PROGRAM MAIN
VAR
	test : UINT;
END_VAR


//DAQ test
//fssf

//daq test

//One

//Two

//Threee


//Four 

//Five

//Six


//Seven

//Eight


//Nine

//Ten

END_PROGRAM

(* stored: Version 1.1.0.1, ProductVersion 3.1.4024.9
   POU MAIN: Id {dd1d77bd-4e25-4335-9864-1fdb214a75d4}, SpecialFunc None *)
